FUNCTION_BLOCK EL2794
VAR
	{attribute addProperty Name "WcState"}
	_wcState : WcStateBase;
	{attribute addProperty Name "Info data"}
	_infoData : InfoDataBase;
	_io : EL2xx4_Data;
END_VAR

PROPERTY IO : REFERENCE TO EL2xx4_Data
GET
IO REF= _io;
END_GET
END_PROPERTY

PROPERTY WcState : REFERENCE TO WcStateBase
GET
WcState REF= _wcState;
END_GET
END_PROPERTY

END_FUNCTION_BLOCK

(* stored: Version 1.1.0.1, ProductVersion 3.1.4024.9
   POU EL2794: Id {205cad7f-67d5-0d4b-1cb2-82bb730c2f44}, SpecialFunc None
   Property IO: Id {644fb6e9-1717-0eab-13ac-a7b1cb30b152}
   Get Get: Id {91b3301b-0d2c-0ecc-3ad7-67affbf5e229}
   Property WcState: Id {f625bbab-4cc8-06d4-2ff1-ca1f068123fb}
   Get Get: Id {539f9204-6775-05fe-1c4c-c25b3c98c7a9} *)
